(* CoDeSys 2.3 project: Nosto_ovi.pro *)
(* Title: Use of different IEC-61131-3 languages *)
(* Version: 1.0.0 *)
(* Author: Niko Siltala (TUT) *)
(* Description: Use of different IEC-61131-3 languages to control a lift door. *)
(* Libraries: STANDARD.LIB 16.8.17 14:08:57 *)

(* Global variable list: Global_Variables *)
VAR_GLOBAL
	I_Limit_Up	: BOOL;	(*Sensor Door limit: Up*)
	I_Limit_Dn	: BOOL;	(*Sensor Door limit: Down*)

	I_Btn_Up	: BOOL;	(*Button: Up*)
	I_Btn_Stop	: BOOL;	(*Button: Stop*)
	I_Btn_Dn	: BOOL;	(*Button: Down*)

	I_Btn_Single	: BOOL;	(*Button: Action*)


	O_Mot_Up	: BOOL;	(*Motor driving Up*)
	O_Mot_Dn	: BOOL;	(*Motor driving Dn*)
END_VAR

(* Data type *)
TYPE E_State :
(
	E_St_Stop_Idle := 0,
	E_St_Drv_Up,
	E_St_Drv_Down
);
END_TYPE

(* POU MAIN_FBD_3Btn, FBD *)
PROGRAM MAIN_FBD_3Btn
VAR
	rs_up: RS;
	rs_dn: RS;
END_VAR
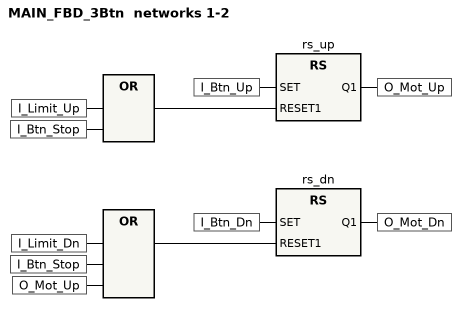
_FBD_ (* Function Block Diagram *)
NETWORK 1
	rs_up:RS(SET: I_Btn_Up, RESET1: OR(I_Limit_Up, I_Btn_Stop)) => O_Mot_Up
NETWORK 2
	rs_dn:RS(SET: I_Btn_Dn, RESET1: OR(I_Limit_Dn, I_Btn_Stop, O_Mot_Up)) => O_Mot_Dn
_END_FBD_
(* the same logic as Structured Text *)
(* Network 1 *)
rs_up(SET := I_Btn_Up, RESET1 := I_Limit_Up OR I_Btn_Stop);
O_Mot_Up := rs_up.Q1;
(* Network 2 *)
rs_dn(SET := I_Btn_Dn, RESET1 := I_Limit_Dn OR I_Btn_Stop OR O_Mot_Up);
O_Mot_Dn := rs_dn.Q1;
END_PROGRAM

(* POU MAIN_LD_3Btn, LD *)
PROGRAM MAIN_LD_3Btn
(*Ks. http://engineeronadisk.com/book_plcs/plc_sequa2.html#16763 for methodologial example*)
VAR
	state	: ARRAY [0..7] OF BOOL;	(*states*)
	tr		: ARRAY [0..7] OF BOOL;	(*transitions*)
	bInitDone: BOOL := FALSE;		(*Intialisation is done*)
END_VAR
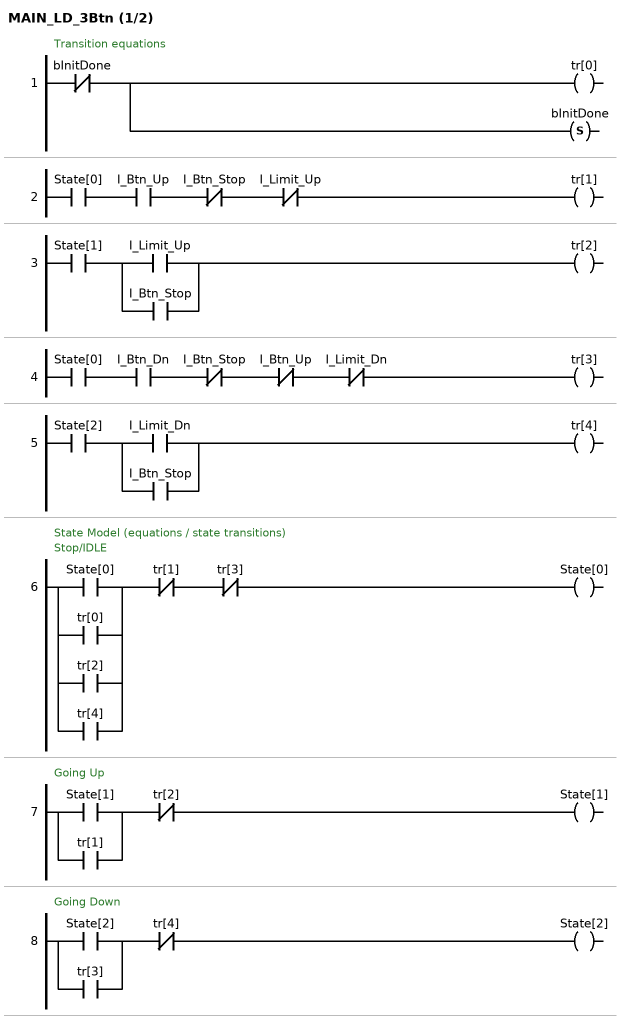
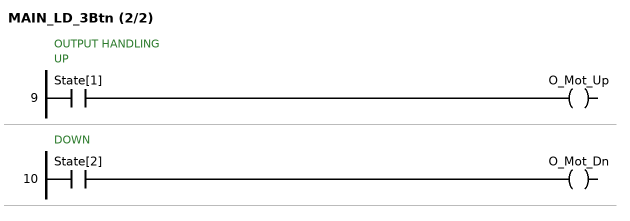
_LD_ (* Ladder Diagram *)
NETWORK 1 (* Transition equations *)
	[/bInitDone] --- (tr[0]) (S bInitDone)
NETWORK 2
	[State[0]] - [I_Btn_Up] - [/I_Btn_Stop] - [/I_Limit_Up] --- (tr[1])
NETWORK 3
	[State[1]] - { [I_Limit_Up] | [I_Btn_Stop] } --- (tr[2])
NETWORK 4
	[State[0]] - [I_Btn_Dn] - [/I_Btn_Stop] - [/I_Btn_Up] - [/I_Limit_Dn] --- (tr[3])
NETWORK 5
	[State[2]] - { [I_Limit_Dn] | [I_Btn_Stop] } --- (tr[4])
NETWORK 6 (* State Model (equations / state transitions) / Stop/IDLE *)
	{ [State[0]] | [tr[0]] | [tr[2]] | [tr[4]] } - [/tr[1]] - [/tr[3]] --- (State[0])
NETWORK 7 (* Going Up *)
	{ [State[1]] | [tr[1]] } - [/tr[2]] --- (State[1])
NETWORK 8 (* Going Down *)
	{ [State[2]] | [tr[3]] } - [/tr[4]] --- (State[2])
NETWORK 9 (* OUTPUT HANDLING / UP *)
	[State[1]] --- (O_Mot_Up)
NETWORK 10 (* DOWN *)
	[State[2]] --- (O_Mot_Dn)
_END_LD_
(* the same logic as Structured Text *)
(* Network 1: Transition equations *)
tr[0] := NOT bInitDone;
IF tr[0] THEN bInitDone := TRUE; END_IF;
(* Network 2 *)
tr[1] := State[0] AND I_Btn_Up AND NOT I_Btn_Stop AND NOT I_Limit_Up;
(* Network 3 *)
tr[2] := State[1] AND (I_Limit_Up OR I_Btn_Stop);
(* Network 4 *)
tr[3] := State[0] AND I_Btn_Dn AND NOT I_Btn_Stop AND NOT I_Btn_Up AND NOT I_Limit_Dn;
(* Network 5 *)
tr[4] := State[2] AND (I_Limit_Dn OR I_Btn_Stop);
(* Network 6: State Model (equations / state transitions) / Stop/IDLE *)
State[0] := (State[0] OR tr[0] OR tr[2] OR tr[4]) AND NOT tr[1] AND NOT tr[3];
(* Network 7: Going Up *)
State[1] := (State[1] OR tr[1]) AND NOT tr[2];
(* Network 8: Going Down *)
State[2] := (State[2] OR tr[3]) AND NOT tr[4];
(* Network 9: OUTPUT HANDLING / UP *)
O_Mot_Up := State[1];
(* Network 10: DOWN *)
O_Mot_Dn := State[2];
END_PROGRAM

(* POU MAIN_SFC_1Btn, SFC *)
PROGRAM MAIN_SFC_1Btn
VAR
	RTrig_Btn	: R_TRIG;	(*Button triggered*)
	tMinStepTime	: TIME	:= t#200ms;
END_VAR
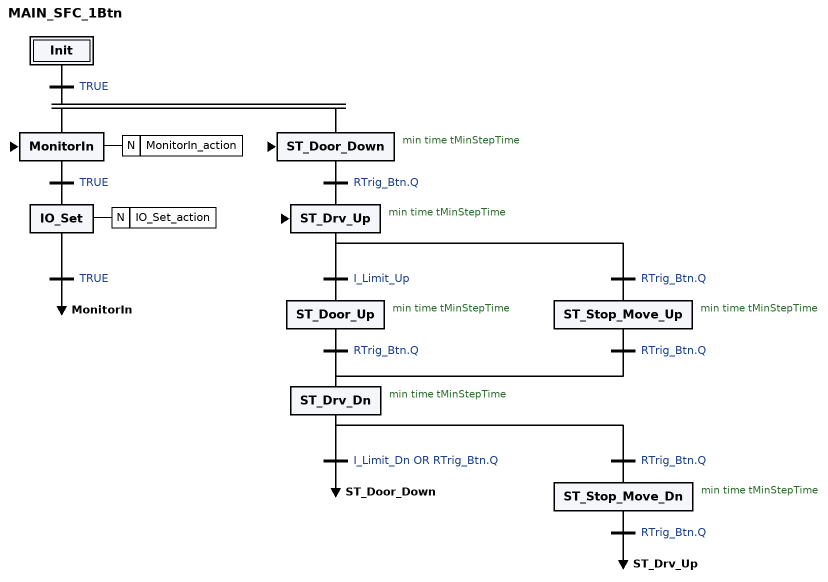
INITIAL_STEP Init:
END_STEP
TRANSITION FROM Init TO (MonitorIn, ST_Door_Down) := TRUE;
END_TRANSITION
STEP MonitorIn:
	MonitorIn_action(N);
END_STEP
TRANSITION FROM MonitorIn TO IO_Set := TRUE;
END_TRANSITION
STEP IO_Set:
	IO_Set_action(N);
END_STEP
TRANSITION FROM IO_Set TO MonitorIn := TRUE;
END_TRANSITION
STEP ST_Door_Down: (* min time tMinStepTime *)
END_STEP
TRANSITION FROM ST_Door_Down TO ST_Drv_Up := RTrig_Btn.Q;
END_TRANSITION
STEP ST_Drv_Up: (* min time tMinStepTime *)
END_STEP
TRANSITION FROM ST_Drv_Up TO ST_Door_Up := I_Limit_Up;
END_TRANSITION
TRANSITION FROM ST_Drv_Up TO ST_Stop_Move_Up := RTrig_Btn.Q;
END_TRANSITION
STEP ST_Stop_Move_Up: (* min time tMinStepTime *)
END_STEP
TRANSITION FROM ST_Stop_Move_Up TO ST_Drv_Dn := RTrig_Btn.Q;
END_TRANSITION
STEP ST_Door_Up: (* min time tMinStepTime *)
END_STEP
TRANSITION FROM ST_Door_Up TO ST_Drv_Dn := RTrig_Btn.Q;
END_TRANSITION
STEP ST_Drv_Dn: (* min time tMinStepTime *)
END_STEP
TRANSITION FROM ST_Drv_Dn TO ST_Door_Down := I_Limit_Dn OR RTrig_Btn.Q;
END_TRANSITION
TRANSITION FROM ST_Drv_Dn TO ST_Stop_Move_Dn := RTrig_Btn.Q;
END_TRANSITION
STEP ST_Stop_Move_Dn: (* min time tMinStepTime *)
END_STEP
TRANSITION FROM ST_Stop_Move_Dn TO ST_Drv_Up := RTrig_Btn.Q;
END_TRANSITION

ACTION MonitorIn_action:
(*Button just pressed*)
RTrig_Btn(CLK:=I_Btn_Single , Q=> );
END_ACTION

ACTION IO_Set_action:
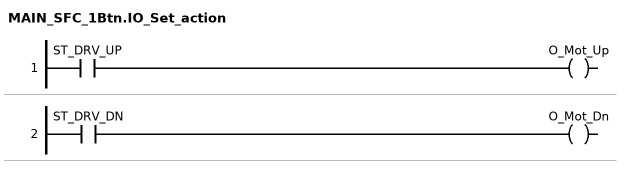
_LD_ (* Ladder Diagram *)
NETWORK 1
	[ST_DRV_UP] --- (O_Mot_Up)
NETWORK 2
	[ST_DRV_DN] --- (O_Mot_Dn)
_END_LD_
(* the same logic as Structured Text *)
(* Network 1 *)
O_Mot_Up := ST_DRV_UP;
(* Network 2 *)
O_Mot_Dn := ST_DRV_DN;
END_ACTION
END_PROGRAM

(* POU MAIN_SFC_3Btn, SFC *)
PROGRAM MAIN_SFC_3Btn
VAR

END_VAR
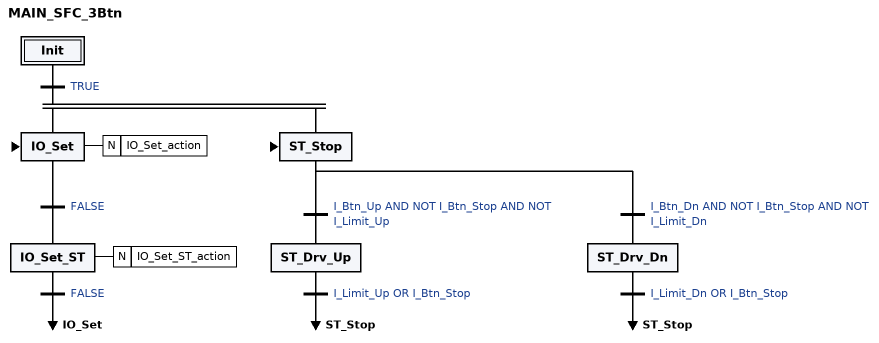
INITIAL_STEP Init:
END_STEP
TRANSITION FROM Init TO (IO_Set, ST_Stop) := TRUE;
END_TRANSITION
STEP IO_Set:
	IO_Set_action(N);
END_STEP
TRANSITION FROM IO_Set TO IO_Set_ST := FALSE;
END_TRANSITION
STEP ST_Stop:
END_STEP
TRANSITION FROM ST_Stop TO ST_Drv_Up := I_Btn_Up AND NOT I_Btn_Stop AND NOT I_Limit_Up;
END_TRANSITION
TRANSITION FROM ST_Stop TO ST_Drv_Dn := I_Btn_Dn AND NOT I_Btn_Stop AND NOT I_Limit_Dn;
END_TRANSITION
STEP ST_Drv_Up:
END_STEP
TRANSITION FROM ST_Drv_Up TO ST_Stop := I_Limit_Up OR I_Btn_Stop;
END_TRANSITION
STEP ST_Drv_Dn:
END_STEP
TRANSITION FROM ST_Drv_Dn TO ST_Stop := I_Limit_Dn OR I_Btn_Stop;
END_TRANSITION
STEP IO_Set_ST:
	IO_Set_ST_action(N);
END_STEP
TRANSITION FROM IO_Set_ST TO IO_Set := FALSE;
END_TRANSITION

ACTION IO_Set_action:
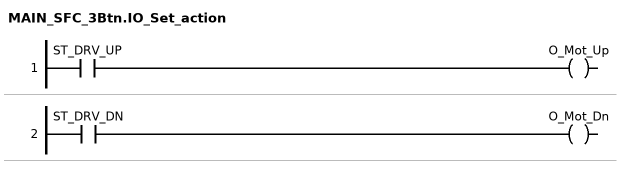
_LD_ (* Ladder Diagram *)
NETWORK 1
	[ST_DRV_UP] --- (O_Mot_Up)
NETWORK 2
	[ST_DRV_DN] --- (O_Mot_Dn)
_END_LD_
(* the same logic as Structured Text *)
(* Network 1 *)
O_Mot_Up := ST_DRV_UP;
(* Network 2 *)
O_Mot_Dn := ST_DRV_DN;
END_ACTION

ACTION IO_Set_ST_action:
(*Updating the outputs*)
O_Mot_Up := ST_DRV_UP;
O_Mot_Dn := ST_DRV_DN;
END_ACTION
END_PROGRAM

(* POU MAIN_ST_3Btn, ST *)
PROGRAM MAIN_ST_3Btn
VAR
	iState			: INT := 0;				(*Current state*)
END_VAR
(*Call the state model and evolve its state.*)
(*Initialise outputs and other variables*)
O_Mot_Up := FALSE;
O_Mot_Dn := FALSE;

(*If stop then always stopped state*)
IF I_Btn_Stop THEN
	iState := 0;
END_IF;

(*Implementation for the state model*)
CASE iState OF
0 :	(*St_Stop_Idle*)
	IF I_Btn_Up AND NOT I_Limit_Up THEN
		iState := 1;
	ELSIF I_Btn_Dn AND NOT I_Limit_Dn THEN
		iState := 2;
	END_IF;

1 :	(*St_Drv_Up*)
	IF I_Limit_Up THEN
		iState := 0;
	END_IF;
	O_Mot_Up := TRUE;

2 : (*St_Drv_Down*)
	IF I_Limit_Dn THEN
		iState := 0;
	END_IF;
	O_Mot_Dn := TRUE;

ELSE
	(*Some odd state change has occurred. Moving into non-defined state -> move to init*)
	iState := 0;
END_CASE;

(*Outputs could be also handled here separately according the state. E.g. with case -statement*)
(*Like this:*)

CASE iState OF
1 :	(*St_Drv_Up*)
	O_Mot_Up := TRUE;

2 : (*St_Drv_Down*)
	O_Mot_Dn := TRUE;

END_CASE;
END_PROGRAM

(* POU MAIN_ST_3Btn_withFB, ST *)
PROGRAM MAIN_ST_3Btn_withFB
VAR
	fbStateModel_3Btn	: FB_StateModel_3Btn;	(*State model implementation*)
	iStateCurr			: E_State;
END_VAR
(*Call the state model and evolve its state.*)
fbStateModel_3Btn(
	iBtn_Up:= I_Btn_Up,
	iBtn_Stop:= I_Btn_Stop,
	iBtn_Dn:= I_Btn_Dn,
	iLimit_Up:= I_Limit_Up,
	iLimit_Dn:= I_Limit_Dn,
	eState_Curr=> iStateCurr,
	bUP=> ,
	bDOWN=> );

(*Resolve and set output states*)
(*Output update - Alternative 1: Using state number/name*)
O_Mot_Up := (fbStateModel_3Btn.eState_Curr = E_St_Drv_Up);
O_Mot_Dn := (fbStateModel_3Btn.eState_Curr = E_St_Drv_Down);

(*Output update - Alternative 2: Using FBs outputs*)
O_Mot_Up := fbStateModel_3Btn.bUP;
O_Mot_Dn := fbStateModel_3Btn.bDOWN;

(*Output update - Alternative 3: Directly capture when calling the instance*)
(*
fbStateModel_3Btn(
	bUP=> O_Mot_Up,
	bDOWN=> O_Mot_Dn); 
*)
END_PROGRAM

(* POU FB_StateModel_3Btn, ST *)
FUNCTION_BLOCK FB_StateModel_3Btn
VAR_INPUT
	iBtn_Up		: BOOL;
	iBtn_Stop	: BOOL;
	iBtn_Dn		: BOOL;
	iLimit_Up	: BOOL;
	iLimit_Dn	: BOOL;
END_VAR
VAR_OUTPUT
	eState_Curr	: E_State;
	bUP 		: BOOL;
	bDOWN		: BOOL;
END_VAR
VAR
	iState 		: E_State	:=0;
END_VAR
bUP:=FALSE;
bDOWN:=FALSE;

(*If stop then always stopped state*)
IF iBtn_Stop THEN
	iState := E_St_Stop_Idle;
END_IF;

CASE iState OF
E_St_Stop_Idle :
	IF iBtn_Up AND NOT I_Limit_Up THEN
		iState := E_St_Drv_Up;
	ELSIF iBtn_Dn AND NOT I_Limit_Dn THEN
		iState := E_St_Drv_Down;
	END_IF;

E_St_Drv_Up :
	IF I_Limit_Up THEN
		iState := E_St_Stop_Idle;
	END_IF;
	bUP:=TRUE;

E_St_Drv_Down :
	IF I_Limit_Dn THEN
		iState := E_St_Stop_Idle;
	END_IF;
	bDOWN := TRUE;

ELSE
	iState := E_St_Stop_Idle;
END_CASE;

eState_Curr := iState;
END_FUNCTION_BLOCK

(* POU Simulator, ST *)
PROGRAM Simulator
VAR
	i 	: INT;
	iDoorPos	: INT;	(*Door position*)
	iDoorPos_Limi_Up	: INT	:= 80;
	iDoorPos_Limi_Dn	: INT	:= -110;
END_VAR
(*Simulate door movement*)
IF O_Mot_Up THEN
	iDoorPos := iDoorPos + 1;
ELSIF O_Mot_Dn THEN
	iDoorPos := iDoorPos - 1;
END_IF;

(*iDoorPos := LIMIT(iDoorPos_Limi_Dn, iDoorPos,iDoorPos_Limi_Up);*)

(*Simulate limit switches*)
IF iDoorPos >= iDoorPos_Limi_Up THEN
	I_Limit_Up := TRUE;
ELSE
	I_Limit_Up := FALSE;
END_IF;

IF iDoorPos <= iDoorPos_Limi_Dn THEN
	I_Limit_Dn := TRUE;
ELSE
	I_Limit_Dn := FALSE;
END_IF;
END_PROGRAM

(* Visualisation VC_1Button
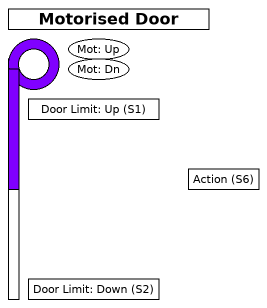
rectangle at (30,90)-(161,111): text "Door Limit: Up (S1)"; alarm colour if .I_Limit_Up; toggles .I_Limit_Up
rectangle at (30,270)-(161,291): text "Door Limit: Down (S2)"; alarm colour if .I_Limit_Dn; toggles .I_Limit_Dn
rounded rectangle at (190,160)-(261,181): text "Action (S6)"; alarm colour if .I_Btn_Single; taps .I_Btn_Single
ellipse at (70,30)-(131,51): text "Mot: Up"; alarm colour if .O_Mot_Up
ellipse at (70,50)-(131,71): text "Mot: Dn"; alarm colour if .O_Mot_Dn
rectangle at (10,0)-(211,21): text "Motorised Door"
rectangle at (10,60)-(21,181): bottom -1*Simulator.iDoorPos
3 more shapes without text or variables
*)

(* Visualisation VC_3Buttons
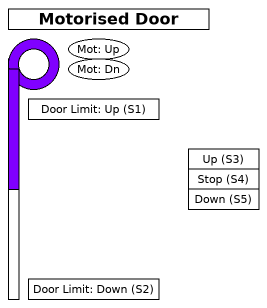
rectangle at (30,90)-(161,111): text "Door Limit: Up (S1)"; alarm colour if .I_Limit_Up; toggles .I_Limit_Up
rectangle at (30,270)-(161,291): text "Door Limit: Down (S2)"; alarm colour if .I_Limit_Dn; toggles .I_Limit_Dn
rounded rectangle at (190,140)-(261,161): text "Up (S3)"; alarm colour if .I_Btn_Up; taps .I_Btn_Up
rounded rectangle at (190,160)-(261,181): text "Stop (S4)"; alarm colour if .I_Btn_Stop; taps .I_Btn_Stop
rounded rectangle at (190,180)-(261,201): text "Down (S5)"; alarm colour if .I_Btn_Dn; taps .I_Btn_Dn
ellipse at (70,30)-(131,51): text "Mot: Up"; alarm colour if .O_Mot_Up
ellipse at (70,50)-(131,71): text "Mot: Dn"; alarm colour if .O_Mot_Dn
rectangle at (10,0)-(211,21): text "Motorised Door"
rectangle at (10,60)-(21,181): bottom -1*Simulator.iDoorPos
3 more shapes without text or variables
*)
